SUBAPPLICATION Heckschieber (* Subapplication Type *)
  (* Standard: 61499-2 *)
  (* Version 1.0, 2023-01-29, Franz *)
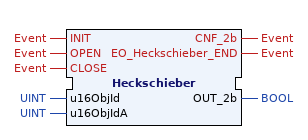
  EVENT_INPUT
    INIT;
    OPEN;
    CLOSE;
  END_EVENT
  EVENT_OUTPUT
    CNF_2b;
    EO_Heckschieber_END;
  END_EVENT
  VAR_INPUT
    u16ObjId : UINT;
    u16ObjIdA : UINT;
  END_VAR
  VAR_OUTPUT
    OUT_2b : BOOL;
  END_VAR
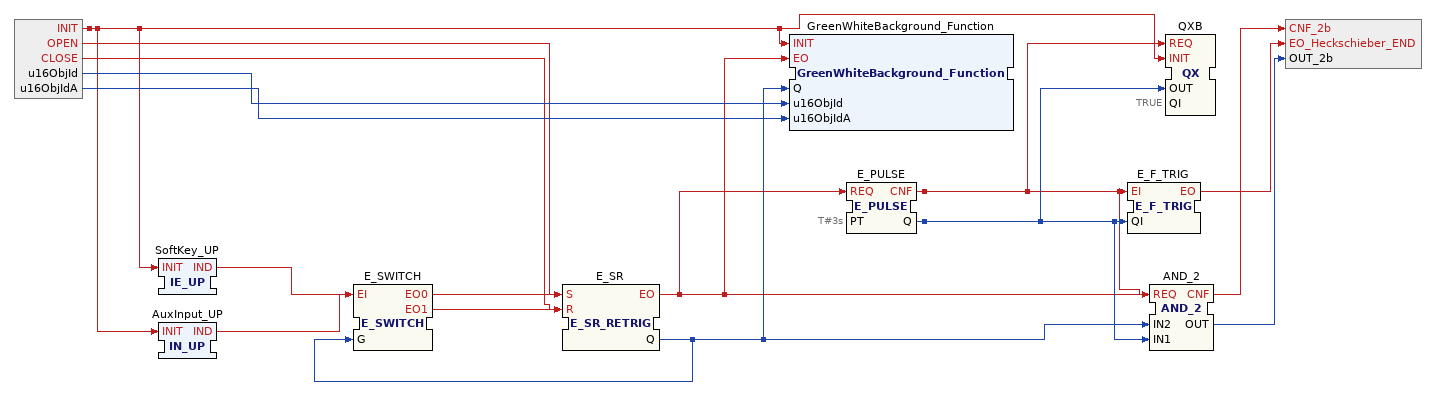
  FBS
    E_F_TRIG : E_F_TRIG;
    QXB : QX(QI := TRUE);
    E_SR : E_SR_RETRIG;
    E_SWITCH : E_SWITCH;
    AND_2 : AND_2;
    E_PULSE : E_PULSE(PT := T#3s);
  END_FBS
  SUBAPPS
    GreenWhiteBackground_Function : GreenWhiteBackground_Function;
    SoftKey_UP : IE_UP;
    AuxInput_UP : IN_UP;
  END_SUBAPPS
  EVENT_CONNECTIONS
    E_PULSE.CNF TO E_F_TRIG.EI;
    E_PULSE.CNF TO QXB.REQ;
    E_SWITCH.EO0 TO E_SR.S;
    E_SWITCH.EO1 TO E_SR.R;
    E_SR.EO TO AND_2.REQ;
    E_SR.EO TO E_PULSE.REQ;
    E_PULSE.CNF TO AND_2.REQ;
    OPEN TO E_SR.S;
    CLOSE TO E_SR.R;
    AND_2.CNF TO CNF_2b;
    E_F_TRIG.EO TO EO_Heckschieber_END;
    INIT TO QXB.INIT;
    INIT TO GreenWhiteBackground_Function.INIT;
    E_SR.EO TO GreenWhiteBackground_Function.EO;
    INIT TO SoftKey_UP.INIT;
    SoftKey_UP.IND TO E_SWITCH.EI;
    INIT TO AuxInput_UP.INIT;
    AuxInput_UP.IND TO E_SWITCH.EI;
  END_CONNECTIONS
  DATA_CONNECTIONS
    E_SR.Q TO E_SWITCH.G;
    E_SR.Q TO AND_2.IN2;
    AND_2.OUT TO OUT_2b;
    E_SR.Q TO GreenWhiteBackground_Function.Q;
    u16ObjId TO GreenWhiteBackground_Function.u16ObjId;
    u16ObjIdA TO GreenWhiteBackground_Function.u16ObjIdA;
    E_PULSE.Q TO E_F_TRIG.QI;
    E_PULSE.Q TO QXB.OUT;
    E_PULSE.Q TO AND_2.IN1;
  END_CONNECTIONS
END_SUBAPPLICATION
